FUNCTION_BLOCK FB_UserLog
VAR_INPUT
	
	nNumberOfData				: DINT;
	bSaveSignal					: BOOL;
	sUser						: STRING;
	sGroup						: STRING;
	sDate						: STRING;
	sTime						: STRING;

END_VAR
VAR_OUTPUT
	
END_VAR
VAR
	rSaveSignal					: R_TRIG;
	i							: DINT;
END_VAR
VAR_IN_OUT
	
	aDataOutput					: ARRAY [*] OF ST_UserLog;
	
END_VAR

rSaveSignal( CLK := bSaveSignal);

IF rSaveSignal.Q THEN
	
	FOR i := nNumberOfData TO 0 BY -1 DO
		
		aDataOutput[i+1]		:= aDataOutput[i];
		
	END_FOR
	
	aDataOutput[0].sDate		:= sDate;
	aDataOutput[0].sGroup		:= sGroup;
	aDataOutput[0].sTime		:= sTime;
	aDataOutput[0].sUser		:= sUser;
	
END_IF

END_FUNCTION_BLOCK

(* stored: Version 1.1.0.1, ProductVersion 3.1.4024.13
   POU FB_UserLog: Id {1570abb7-f10f-4062-98c8-8686e7ab373c}, SpecialFunc None *)
